FUNCTION_BLOCK BOOL_Param
VAR_INPUT PERSISTENT
	val				: BOOL;
END_VAR

END_FUNCTION_BLOCK

(* stored: Version 1.1.0.1
   POU BOOL_Param: Id {86d3985b-ce36-49e3-b31b-ca03b5ee72a3}, SpecialFunc None *)
